FUNCTION_BLOCK FB_FanControl
VAR
//-----PWM-----
	uiPwmPeriod					AT %Q*	:UINT :=40;				//PWMの周期,μｓ単位で、FANは25Hz入力なので、40μs設定
	uiPwmOutput					AT %Q*	:UINT :=65535;			//PWMのパルス幅、％単位の入力。初期値はMAX値(100%)を入力
	_rMaxTemp							:REAL;					//PWMのパルス幅を100%にする温度
	_rMinTemp							:REAL;					//PWMのパルス幅を0%にする温度
	_bManualFanSpeed					:BOOL;					//FANマニュアルスピード有効
	_uiManualFanSpeed					:UINT;					//FANマニュアルスピード設定

//-----吸気ファン-----
	bInFanOn					AT %Q*	:BOOL :=TRUE;			//吸気ファン運転、基本回っているように初期値はTRUE
	_iInAirTemp					AT %I*	:INT;					//吸気ファン側の測温抵抗体温度
	usiInFanInputEvent			AT %I*	:USINT;					//入力が500μs中に何回あったか
	udiInFanInputEventTime		AT %I*	:ARRAY[1..10] OF UDINT;	//入力があった時間
	udiInFanPrevEventTime				:UDINT;					//入力があった前回の時間
	udiInFanDeltaTime					:UDINT;					//入力時間の差
	iInFanInputEventCountUp				:INT;					//入力回数をカウント
	_rInFanSpeed						:REAL;					//吸気ファンの回転スピード[rpm]

//-----排気ファン-----
	bOutFanOn					AT %Q*	:BOOL :=TRUE;			//排気ファン運転、基本回っているように初期値はTRUE	
	_iOutAirTemp				AT %I*	:INT;					//排気ファン側の測温抵抗体温度	
	usiOutFanInputEvent			AT %I*	:USINT;					//入力が500μs中に何回あったか
	udiOutFanInputEventTime		AT %I*	:ARRAY[1..10] OF UDINT;	//入力があった時間
	udiOutFanPrevEventTime				:UDINT;					//入力があった前回の時間
	udiOutFanDeltaTime					:UDINT;					//入力時間の差
	iOutFanInputEventCountUp			:INT;					//入力回数をカウント
	_rOutFanSpeed						:REAL;					//排気ファンの回転スピード[rpm]	
	
END_VAR

(*
FANの仕様
メーカー：オリエンタルモーター
型番：MDV925-24S
電圧：24V
電流：0.04A-0.20A(PWMデューティ0%-100%)
回転速度:1500rpm-5000rpm(PWMデューティ0%-100%)

PWM仕様
PWMデューティ比 (％) ＝ TH/T ×100
PWM 周波数25 (kHz) ＝ 1/T


パルスセンサ
1回転あたり2周期の矩形波の信号を出力するセンサです。回転速度の検出ができます。

パルス入力の仕様
ns単位の32bitでタイムスタンプは与えられる
なので、60s中にパルス数で回転数になるので、60.000,000,000nsを,1回転当たり2周期の信号がFANから出力されるので、５回分のタイムスタンプ差のデルタタイムで割り算する


T1℃の時にパルス幅を0%、T2℃の時にパルス幅100%になるように数式作成
y軸をパルス幅に設定、x軸を温度に設定
y=(dパルス幅/d温度)*x+b
y=(100/(T2-T1))*x+b
0=(100/(T2-T1))*T1+b
b=-100*T1/(T2-T1)

y=100*(x-T1)/(T2-T1)
*)

METHOD AirFanOn
VAR_INPUT
END_VAR
//-----ファンの回転数を計算-----
	//吸気ファン
	_rInFanSpeed:=FC_FanSpeedCalc(	usiFanInputEvent		:=usiInFanInputEvent,
									udiFanInputEventTime	:=udiInFanInputEventTime,
									udiFanPrevEventTime		:=udiInFanPrevEventTime,
									udiFanDeltaTime			:=udiInFanDeltaTime,
									iFanInputEventCountUp	:=iInFanInputEventCountUp);
	//排気ファン
	_rOutFanSpeed:=FC_FanSpeedCalc(	usiFanInputEvent		:=usiOutFanInputEvent,
									udiFanInputEventTime	:=udiOutFanInputEventTime,
									udiFanPrevEventTime		:=udiOutFanPrevEventTime,
									udiFanDeltaTime			:=udiOutFanDeltaTime,
									iFanInputEventCountUp	:=iOutFanInputEventCountUp);

//-----測温抵抗体の温度からPWMの出力幅を決定,マニュアルスピードの場合はマニュアルスピードに変更-----
	IF _bManualFanSpeed=TRUE THEN
		uiPwmOutput:=_uiManualFanSpeed;
	ELSIF _rMaxTemp-_rMinTemp<>0 THEN
		uiPwmOutput:=LREAL_TO_UINT(65535*(_iOutAirTemp/10-_rMinTemp)/(_rMaxTemp-_rMinTemp));
	END_IF
END_METHOD

PROPERTY bManualFanSpeed : BOOL
SET
_bManualFanSpeed:=bManualFanSpeed;
END_SET
END_PROPERTY

METHOD PRIVATE FC_FanSpeedCalc : REAL
VAR_INPUT
	usiFanInputEvent				:USINT;							//入力が500μs中に何回あったか
	udiFanInputEventTime			:ARRAY[1..10] OF UDINT;			//入力があった時間
	udiFanPrevEventTime				:REFERENCE TO UDINT;			//入力があった前回の時間
	udiFanDeltaTime					:REFERENCE TO UDINT;			//入力時間の差	
	iFanInputEventCountUp			:REFERENCE TO INT;				//入力回数をカウント
END_VAR
//-----ファンの回転数を計算-----
	CASE usiFanInputEvent OF
		0:
			(*NA*)
		
		1..4:
			IF iFanInputEventCountUp+usiFanInputEvent<=4 THEN
				iFanInputEventCountUp:=iFanInputEventCountUp+usiFanInputEvent;
				
			ELSE
				IF udiFanInputEventTime[5-iFanInputEventCountUp]>udiFanPrevEventTime THEN
					udiFanDeltaTime:=udiFanInputEventTime[5-iFanInputEventCountUp]-udiFanPrevEventTime;
				END_IF
				udiFanPrevEventTime:=udiFanInputEventTime[usiFanInputEvent];
				
				iFanInputEventCountUp:=1;	
				
			END_IF

			
		5..10:
			udiFanDeltaTime:=udiFanInputEventTime[5]-udiFanInputEventTime[1];

			udiFanPrevEventTime:=udiFanInputEventTime[usiFanInputEvent];
			
			iFanInputEventCountUp:=1;
		
	END_CASE
	
	IF udiFanDeltaTime<>0 THEN
		FC_FanSpeedCalc:=60000000000.0/UDINT_TO_REAL(udiFanDeltaTime);
	END_IF
END_METHOD

PROPERTY iInAirTemp : INT
GET
iInAirTemp:=_iInAirTemp;
END_GET
END_PROPERTY

PROPERTY iOutAirTemp : INT
GET
iOutAirTemp:=_iOutAirTemp;
END_GET
END_PROPERTY

PROPERTY rInFanSpeed : REAL
GET
rInFanSpeed:=_rInFanSpeed;
END_GET
END_PROPERTY

PROPERTY rMaxTemp : REAL
SET
_rMaxTemp:=rMaxTemp;
END_SET
END_PROPERTY

PROPERTY rMinTemp : REAL
SET
_rMinTemp:=rMinTemp;
END_SET
END_PROPERTY

PROPERTY rOutFanSpeed : REAL
GET
rOutFanSpeed:=_rOutFanSpeed;
END_GET
END_PROPERTY

PROPERTY uiManualFanSpeed : UINT
SET
_uiManualFanSpeed:=uiManualFanSpeed;
END_SET
END_PROPERTY

END_FUNCTION_BLOCK

(* stored: Version 1.1.0.1, ProductVersion 3.1.4026.12
   POU FB_FanControl: Id {9af4c240-540e-4619-afae-ff9d8bbe47d5}, SpecialFunc None
   Method AirFanOn: Id {8d6735c8-a6eb-41a1-aef6-e6d4faca0110}
   Property bManualFanSpeed: Id {66f76369-2db0-4299-82df-ececf334efd7}
   Set Set: Id {7d16de46-b1eb-4f1d-848f-8167e4af1268}
   Method FC_FanSpeedCalc: Id {c125ef6a-e83d-4b93-a688-90e241b65c85}
   Property iInAirTemp: Id {47fa03f2-3e3f-4d02-b889-7c7078da03b3}
   Get Get: Id {e5858e55-a93c-4e0f-a34d-116f8a4a4a2b}
   Property iOutAirTemp: Id {e537b060-acd0-4cf8-b640-98204ebc554e}
   Get Get: Id {5fdf0e38-f3da-404c-85e1-b0260da7e066}
   Property rInFanSpeed: Id {88542c56-0b72-466c-971c-00018d548bfb}
   Get Get: Id {d6ce33bb-5ce6-4170-bd1d-b5c8f9fbcd62}
   Property rMaxTemp: Id {41853c5c-4a0d-4ef0-8a4a-14c3c10af275}
   Set Set: Id {1df49628-980f-4fc2-9ead-fd57232bfff5}
   Property rMinTemp: Id {26f67bdc-9975-4005-aa80-3238059ba1c1}
   Set Set: Id {e3a2c8af-c300-4de5-9c8f-09e7ac67acfa}
   Property rOutFanSpeed: Id {af9fa307-1268-49c6-a92f-dad8658a07bb}
   Get Get: Id {de0dc0cd-fb69-4984-82ba-658e108ffde5}
   Property uiManualFanSpeed: Id {3099676e-f9f9-4245-8b49-4a1f8c0dc16b}
   Set Set: Id {a3ef9020-c18d-4397-b816-af4e848e49a9} *)
